Staubli VAL3: subString.pgx

public program subString(string& x_sInput[], num x_nStart, num x_nEnd, string& x_sResult[])
  local num l_nElement
  local num l_nLength
begin

  l_nLength = size(x_sInput)
  resize(x_sResult,1,1)
  x_sResult =""
  resize(x_sResult,1,l_nLength)

  // iterate complete input x_sInput[0] ... x_sInput[l_nLength-1]
  for l_nElement = 0 to l_nLength-1

    x_sResult[l_nElement] = mid(x_sInput[l_nElement], x_nEnd-x_nStart+1,x_nStart)

  endFor

end
